// TwinCAT 3 PLC project Twingrind
// Title: Twingrind
// Company: Stefan Besler
// Author: Stefan Besler and Contributers
// ProjectVersion: 0.4.1.0
// ProgramVersion: 3.1.4023.0
// libraries:
//   Tc2_Standard, * (Beckhoff Automation GmbH)
//   Tc2_System, * (Beckhoff Automation GmbH)
// project tree:
//   / CaptureMode.TcDUT, Profiler.TcPOU, ParameterList.TcGVL, FrameData.TcDUT, FrameMeta.TcDUT

// ---- CaptureMode.TcDUT
{attribute 'qualified_only'}
{attribute 'strict'}
TYPE CaptureMode :
(
	All, //< Capture all callstacks if the data array is full, old entries are overwritten
  Fastest, //< Capture only the fastest callstacks, data of slower callstacks are overwritten
  Slowest, //< Capture only the slowest callstacks, data of faster callstacks are overwritten
  FirstOnesOnly //< Only capture callstacks until the data array is not completely full
);
END_TYPE

// ---- FrameData.TcDUT
TYPE INTERNAL FrameData :
STRUCT
  Hash : UDINT;
  Depth : DINT;
  StartLo : DWORD;
  StartHi : DWORD;  
  EndLo : DWORD;
  EndHi : DWORD;  
END_STRUCT
END_TYPE

// ---- FrameMeta.TcDUT
TYPE INTERNAL FrameMeta :
STRUCT
  {attribute 'displaymode':='hex'}
  Id : UDINT;
  Size : DINT;
  TotalDuration : LWORD; 
END_STRUCT
END_TYPE

// ---- ParameterList.TcGVL
{attribute 'qualified_only'}
VAR_GLOBAL CONSTANT
  MAX_FRAMES : SINT := 10; //< Maximum number of callstacks that can be captured by the profiler. Note that CaptureMode controls how and if old frames are overwritten by the profiler
  MAX_STACKSIZE : DINT := 32000*10; //< Storage buffer for calls within a cycle. Every call uses 2 entries. Adjust this value if you use loads of methods in your PLC
END_VAR

// ---- Profiler.TcPOU
{attribute 'hide_all_locals'}
PROGRAM Profiler
VAR_INPUT
  CaptureOnce : BOOL; //< On rising edge, starts to one frame
  CaptureContinuous : BOOL; //<  If set record until all frames are filled up, [MAX_FRAMES](xref:Profiler.ParameterList#MAX_FRAMES) controls how many frames are recorded. If all frames are recorded, the flag is reset
  Mode : CaptureMode;
  CaptureCpuTimeLowThreshold : LREAL; //< In percent (0 - 100) to controls the minimum cycletime that frame need to have in order to be recorded, if CaptureCpuTimeLowThreshold = CaptureCpuTimeHighThreshold = 0, all frame are recorded
  CaptureCpuTimeHighThreshold : LREAL; //< In percent (0 - 100) to controls the maximum cycletime that frame need to have in order to be recorded  
  Reset : BOOL; //< On rising edge, deletes all recorded frames
END_VAR
VAR_OUTPUT
  Busy : BOOL;
  Error : BOOL;
  ErrorMessage : STRING;
  FrameIndex : SINT;  
  Meta : ARRAY [0..ParameterList.MAX_FRAMES] OF FrameMeta;
  Data : ARRAY [0..ParameterList.MAX_FRAMES, 1..MAX_TASKS] OF ARRAY[0..ParameterList.MAX_STACKSIZE] OF FrameData;
  CycleTime : ARRAY [1..MAX_TASKS] OF UDINT; //< Cycletime for every task in 100ns
  Tasks : SINT;
END_VAR
VAR
  _size : DINT;
  _meta : REFERENCE TO FrameMeta REF= Meta[0];
  _data : REFERENCE TO ARRAY[0..ParameterList.MAX_STACKSIZE] OF FrameData REF= Data[0, 1];
  _cpuCounter : GETCPUCOUNTER;
  _currenttask : GETCURTASKINDEX;
  _cycleDuration : LREAL; //< in percent
  _enabled : BOOL;
  _maxDuration : LREAL;
  _depth : DINT := 0;
  _frameRecorded : F_TRIG;
  _captureOnceTrig : R_TRIG;
  _captureContinuousTrig : R_TRIG;
  _resetTrig : R_TRIG;
  _i, _j : SINT;
  _taskIt : UDINT;
END_VAR
VAR CONSTANT
  MAX_TASKS : SINT:=1;
END_VAR

_enabled := FALSE;
_frameRecorded(CLK:=_enabled);
_captureOnceTrig(CLK:=CaptureOnce);
_resetTrig(CLK:=Reset);
_captureContinuousTrig(CLK:=CaptureContinuous);

// Initialization get cycle time for all tasks. Report an
// error if the PLC is using more than 1 task, because this is not
// supported atm
IF _taskIt < 1
THEN
  IF TwinCAT_SystemInfoVarList._AppInfo.TaskCnt > SINT_TO_UDINT(MAX_TASKS)
  THEN
    Error := TRUE;
    ErrorMessage := 'Twingrind only supports PLCs with 1 tasks only!';
    RETURN;
	END_IF
  
  Tasks := UDINT_TO_SINT(TwinCAT_SystemInfoVarList._AppInfo.TaskCnt);
  FOR _taskIt:=1 TO TwinCAT_SystemInfoVarList._AppInfo.TaskCnt
  DO
    CycleTime[_taskIt] := TwinCAT_SystemInfoVarList._TaskInfo[_taskIt].CycleTime;
	END_FOR
END_IF

IF _captureContinuousTrig.Q
THEN
  CaptureOnce := 0;
  Error := FALSE;
  ErrorMessage := '';
END_IF

// Logic to only keep frames that satisfy the threshold conditions
IF _frameRecorded.Q
THEN
  _meta.Size := _size;
  _meta.TotalDuration := _data[_size-1].EndHi - _data[0].StartHi + _data[_size-1].EndLo - _data[0].StartLo;
  _currenttask();
  
  // Check if the frame that was just recorded should be kept, if so, find the next place in the date structure where
  // we can write into
  _cycleDuration := 100 * UDINT_TO_LREAL(TwinCAT_SystemInfoVarList._TaskInfo[_currenttask.index].LastExecTime) / UDINT_TO_LREAL(TwinCAT_SystemInfoVarList._TaskInfo[_currenttask.index].CycleTime);
  IF (_cycleDuration > CaptureCpuTimeLowThreshold AND_THEN _cycleDuration < CaptureCpuTimeHighThreshold) OR_ELSE 
     (CaptureCpuTimeLowThreshold = 0 AND_THEN CaptureCpuTimeHighThreshold = 0)
  THEN
    FrameIndex := NextFrameIndex();
  END_IF

END_IF

IF CaptureContinuous
THEN
  _enabled := TRUE;
  _size := 0;
ELSE
  IF _captureOnceTrig.Q
  THEN
    Error := FALSE;
    ErrorMessage := '';
    _enabled := TRUE;
    _size := 0;
  END_IF 
END_IF

// Delete all Ddata that has already been caputured
IF _resetTrig.Q
THEN
  Error := FALSE;
  ErrorMessage := '';
  FrameIndex := 0;
  MEMSET(ADR(Data), 0, SIZEOF(Data));
  MEMSET(ADR(Meta), 0, SIZEOF(Meta));
  _enabled := FALSE;
END_IF

// Prepare the current frame
Busy := _enabled;
_depth := 0;
_data REF= Data[FrameIndex, 1];
_meta REF= Meta[FrameIndex];
_meta.Id := TwinCAT_SystemInfoVarList._TaskInfo[1].CycleCount;
_frameRecorded(CLK:=_enabled);

METHOD INTERNAL NextFrameIndex : SINT
VAR
  i : SINT;
  duration : LWORD;
END_VAR
CASE Mode
OF
  // Find the index of the fastest profile
  CaptureMode.Slowest:
    duration := 0;
    FOR i:=0 TO ParameterList.MAX_FRAMES
    DO
      IF Meta[i].TotalDuration = 0
      THEN
        NextFrameIndex := i;
        RETURN;
      ELSIF Meta[i].TotalDuration < duration OR_ELSE duration = 0
      THEN
        duration := Meta[i].TotalDuration;
        NextFrameIndex := i;
      END_IF
    END_FOR

  // Record all frames, just get the next frame index
  CaptureMode.All:
    NextFrameIndex := FrameIndex + 1;
    IF NextFrameIndex > ParameterList.MAX_FRAMES
    THEN
      NextFrameIndex := 0;
    END_IF

  // Find the index of the slowest profile
  CaptureMode.Fastest:
    duration := 0;
    FOR i:=0 TO ParameterList.MAX_FRAMES
    DO
      IF Meta[i].TotalDuration = 0
      THEN
        NextFrameIndex := i;
        RETURN;
      ELSIF Meta[i].TotalDuration > duration OR_ELSE duration = 0
      THEN
        duration := Meta[i].TotalDuration;
        NextFrameIndex := i;
      END_IF
    END_FOR

  // Only record max_frames, then no further frames are caputured
  CaptureMode.FirstOnesOnly:
    NextFrameIndex := MIN(FrameIndex + 1, ParameterList.MAX_FRAMES);

END_CASE
END_METHOD

METHOD Pop
VAR_INPUT
  hash : UDINT;
END_VAR
IF NOT _enabled
THEN
  RETURN;
END_IF

_depth := _depth - 1;
_data[_size].Depth := _depth;
_data[_size].Hash := hash;
_data[_size].StartHi := 0;
_data[_size].StartLo := 0;
_cpuCounter(cpuCntLoDW => _data[_size].EndLo, cpuCntHiDW => _data[_size].EndHi);

IF _depth < 0
THEN
  _enabled := FALSE;
  Error := TRUE;
  ErrorMessage := 'Pop/Push mismatch!';
  RETURN;   
ELSE
  _size := _size + 1;
END_IF

// abort if the stack is getting too big (too many functions were called)
IF _size > ParameterList.MAX_STACKSIZE
THEN
  _enabled := FALSE;
  Error := TRUE;
  ErrorMessage := 'The method stack is too big!';  
END_IF
END_METHOD

METHOD Push
VAR_INPUT
  hash : UDINT;
END_VAR
IF NOT _enabled
THEN
  RETURN;
END_IF

_data[_size].depth := _depth;
_data[_size].hash := hash;
_cpuCounter(cpuCntLoDW => _data[_size].StartLo, cpuCntHiDW => _data[_size].StartHi);
_data[_size].endhi := 0;
_data[_size].endlo := 0;
_size := _size + 1;
_depth := _depth + 1;

// abort if the stack is getting too big (too many functions were called)
IF _size > ParameterList.MAX_STACKSIZE
THEN
  _enabled := FALSE;
  Error := TRUE;
  ErrorMessage := 'The method stack is too big!';
END_IF
END_METHOD

END_PROGRAM
